(* Logix 5000 project; controller project2 vendor 1 type 14 code 54 rev 20.19; software revision 20.05 *)

TASK MainTask (continuous, watchdog 500 ms) : MainProgram

MODULES
   Local : vendor 1 type 14 code 54 (ICP 0, rev 20.19)
      fifth_module : 1756-OB32 (ICP 5, rev 3.2, Output RPI 20 ms)
END_MODULES

VAR_GLOBAL   (* controller tags *)
   TAG_1_CONT : DINT;
END_VAR

PROGRAM MainProgram   (* main routine MainRoutine *)
VAR
   TAG_1_P_MAIN : DINT;
   TAG_2_P_MAIN : DINT;
END_VAR

ROUTINE MainRoutine   (* ladder *)
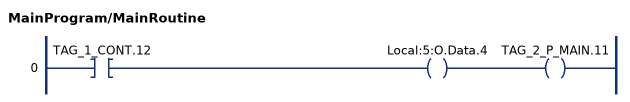
   0: XIC(TAG_1_CONT.12)OTE(Local:5:O.Data.4)OTE(TAG_2_P_MAIN.11);
END_ROUTINE
END_PROGRAM
